(* IEC 61131-3 sources: volt/packages/volt-lsp-iec/test-corpus/lenze-mid/Device/Plc Logic/Application/Library Manager/(unresolved)/cmpopcuastack interfaces, 277 files *)

(* ---- OPCUA_ACTIVATESESSIONREQUEST.dut ---- *)
TYPE OPCUA_ACTIVATESESSIONREQUEST :
STRUCT
	REQUESTHEADER : OpcUa_RequestHeader;
	CLIENTSIGNATURE : OpcUa_SignatureData;
	NOOFCLIENTSOFTWARECERTIFICATES : OpcUa_Int32;
	CLIENTSOFTWARECERTIFICATES : POINTER TO OpcUa_SignedSoftwareCertificate;
	NOOFLOCALEIDS : OpcUa_Int32;
	LOCALEIDS : POINTER TO OpcUa_String;
	USERIDENTITYTOKEN : OpcUa_ExtensionObject;
	USERTOKENSIGNATURE : OpcUa_SignatureData;
END_STRUCT
END_TYPE

(* ---- OPCUA_ACTIVATESESSIONRESPONSE.dut ---- *)
TYPE OPCUA_ACTIVATESESSIONRESPONSE :
STRUCT
	RESPONSEHEADER : OpcUa_ResponseHeader;
	SERVERNONCE : OpcUa_ByteString;
	NOOFRESULTS : OpcUa_Int32;
	RESULTS : POINTER TO OpcUa_StatusCode;
	NOOFDIAGNOSTICINFOS : OpcUa_Int32;
	DIAGNOSTICINFOS : POINTER TO OpcUa_DiagnosticInfo;
END_STRUCT
END_TYPE

(* ---- OPCUA_ADDNODESITEM.dut ---- *)
TYPE OPCUA_ADDNODESITEM :
STRUCT
	PARENTNODEID : OpcUa_ExpandedNodeId;
	REFERENCETYPEID : OpcUa_NodeId;
	REQUESTEDNEWNODEID : OpcUa_ExpandedNodeId;
	BROWSENAME : OpcUa_QualifiedName;
	NODECLASS : OpcUa_NodeClass;
	NODEATTRIBUTES : OpcUa_ExtensionObject;
	TYPEDEFINITION : OpcUa_ExpandedNodeId;
END_STRUCT
END_TYPE

(* ---- OPCUA_ADDNODESREQUEST.dut ---- *)
TYPE OPCUA_ADDNODESREQUEST :
STRUCT
	REQUESTHEADER : OpcUa_RequestHeader;
	NOOFNODESTOADD : OpcUa_Int32;
	NODESTOADD : POINTER TO OpcUa_AddNodesItem;
END_STRUCT
END_TYPE

(* ---- OPCUA_ADDNODESRESPONSE.dut ---- *)
TYPE OPCUA_ADDNODESRESPONSE :
STRUCT
	RESPONSEHEADER : OpcUa_ResponseHeader;
	NOOFRESULTS : OpcUa_Int32;
	RESULTS : POINTER TO OpcUa_AddNodesResult;
	NOOFDIAGNOSTICINFOS : OpcUa_Int32;
	DIAGNOSTICINFOS : POINTER TO OpcUa_DiagnosticInfo;
END_STRUCT
END_TYPE

(* ---- OPCUA_ADDNODESRESULT.dut ---- *)
TYPE OPCUA_ADDNODESRESULT :
STRUCT
	STATUSCODE : OpcUa_StatusCode;
	ADDEDNODEID : OpcUa_NodeId;
END_STRUCT
END_TYPE

(* ---- OPCUA_ADDREFERENCESITEM.dut ---- *)
TYPE OPCUA_ADDREFERENCESITEM :
STRUCT
	SOURCENODEID : OpcUa_NodeId;
	REFERENCETYPEID : OpcUa_NodeId;
	ISFORWARD : OpcUa_Boolean;
	TARGETSERVERURI : OpcUa_String;
	TARGETNODEID : OpcUa_ExpandedNodeId;
	TARGETNODECLASS : OpcUa_NodeClass;
END_STRUCT
END_TYPE

(* ---- OPCUA_ADDREFERENCESREQUEST.dut ---- *)
TYPE OPCUA_ADDREFERENCESREQUEST :
STRUCT
	REQUESTHEADER : OpcUa_RequestHeader;
	NOOFREFERENCESTOADD : OpcUa_Int32;
	REFERENCESTOADD : POINTER TO OpcUa_AddReferencesItem;
END_STRUCT
END_TYPE

(* ---- OPCUA_ADDREFERENCESRESPONSE.dut ---- *)
TYPE OPCUA_ADDREFERENCESRESPONSE :
STRUCT
	RESPONSEHEADER : OpcUa_ResponseHeader;
	NOOFRESULTS : OpcUa_Int32;
	RESULTS : POINTER TO OpcUa_StatusCode;
	NOOFDIAGNOSTICINFOS : OpcUa_Int32;
	DIAGNOSTICINFOS : POINTER TO OpcUa_DiagnosticInfo;
END_STRUCT
END_TYPE

(* ---- OPCUA_AGGREGATECONFIGURATION.dut ---- *)
TYPE OPCUA_AGGREGATECONFIGURATION :
STRUCT
	USESERVERCAPABILITIESDEFAULTS : OpcUa_Boolean;
	TREATUNCERTAINASBAD : OpcUa_Boolean;
	PERCENTDATABAD : OpcUa_Byte;
	PERCENTDATAGOOD : OpcUa_Byte;
	USESLOPEDEXTRAPOLATION : OpcUa_Boolean;
END_STRUCT
END_TYPE

(* ---- OPCUA_AGGREGATEFILTER.dut ---- *)
TYPE OPCUA_AGGREGATEFILTER :
STRUCT
	STARTTIME : OpcUa_DateTime;
	AGGREGATETYPE : OpcUa_NodeId;
	PROCESSINGINTERVAL : OpcUa_Double;
	AGGREGATECONFIGURATION : OpcUa_AggregateConfiguration;
END_STRUCT
END_TYPE

(* ---- OPCUA_AGGREGATEFILTERRESULT.dut ---- *)
TYPE OPCUA_AGGREGATEFILTERRESULT :
STRUCT
	REVISEDSTARTTIME : OpcUa_DateTime;
	REVISEDPROCESSINGINTERVAL : OpcUa_Double;
	REVISEDAGGREGATECONFIGURATION : OpcUa_AggregateConfiguration;
END_STRUCT
END_TYPE

(* ---- OPCUA_ANNOTATION.dut ---- *)
TYPE OPCUA_ANNOTATION :
STRUCT
	MESSAGE : OpcUa_String;
	USERNAME : OpcUa_String;
	ANNOTATIONTIME : OpcUa_DateTime;
END_STRUCT
END_TYPE

(* ---- OPCUA_ANONYMOUSIDENTITYTOKEN.dut ---- *)
TYPE OPCUA_ANONYMOUSIDENTITYTOKEN :
STRUCT
	POLICYID : OpcUa_String;
END_STRUCT
END_TYPE

(* ---- OPCUA_APPLICATIONDESCRIPTION.dut ---- *)
TYPE OPCUA_APPLICATIONDESCRIPTION :
STRUCT
	APPLICATIONURI : OpcUa_String;
	PRODUCTURI : OpcUa_String;
	APPLICATIONNAME : OpcUa_LocalizedText;
	APPLICATIONTYPE : OpcUa_ApplicationType;
	GATEWAYSERVERURI : OpcUa_String;
	DISCOVERYPROFILEURI : OpcUa_String;
	NOOFDISCOVERYURLS : OpcUa_Int32;
	DISCOVERYURLS : POINTER TO OpcUa_String;
END_STRUCT
END_TYPE

(* ---- OPCUA_APPLICATIONTYPE.dut ---- *)
TYPE OPCUA_APPLICATIONTYPE :
(
	OPCUA_APPLICATIONTYPE_SERVER := 0,
	OPCUA_APPLICATIONTYPE_CLIENT := 1,
	OPCUA_APPLICATIONTYPE_CLIENTANDSERVER := 2,
	OPCUA_APPLICATIONTYPE_DISCOVERYSERVER := 3
);
END_TYPE

(* ---- OPCUA_ARGUMENT.dut ---- *)
TYPE OPCUA_ARGUMENT :
STRUCT
	NAME : OpcUa_String;
	DATATYPE : OpcUa_NodeId;
	VALUERANK : OpcUa_Int32;
	NOOFARRAYDIMENSIONS : OpcUa_Int32;
	ARRAYDIMENSIONS : POINTER TO OpcUa_UInt32;
	DESCRIPTION : OpcUa_LocalizedText;
END_STRUCT
END_TYPE

(* ---- OPCUA_ARRAYTYPE.dut ---- *)
TYPE OPCUA_ARRAYTYPE :
(
	OPCUA_VALUERANKS_SCALARORONEDIMENSION := -3,
	OPCUA_VALUERANKS_ANY := -2,
	OPCUA_VALUERANKS_SCALAR := -1,
	OPCUA_VALUERANKS_ONEORMOREDIMENSIONS := 0,
	OPCUA_VALUERANKS_ONEDIMENSION := 1,
	OPCUA_VALUERANKS_TWODIMENSIONS := 2
);
END_TYPE

(* ---- OPCUA_ATTRIBUTEOPERAND.dut ---- *)
TYPE OPCUA_ATTRIBUTEOPERAND :
STRUCT
	NODEID : OpcUa_NodeId;
	ALIAS : OpcUa_String;
	BROWSEPATH : OpcUa_RelativePath;
	ATTRIBUTEID : OpcUa_UInt32;
	INDEXRANGE : OpcUa_String;
END_STRUCT
END_TYPE

(* ---- OPCUA_ATTRIBUTES.dut ---- *)
TYPE OPCUA_ATTRIBUTES :
(
	OPCUA_ATTRIBUTES_NODEID := 1,
	OPCUA_ATTRIBUTES_NODECLASS := 2,
	OPCUA_ATTRIBUTES_BROWSENAME := 3,
	OPCUA_ATTRIBUTES_DISPLAYNAME := 4,
	OPCUA_ATTRIBUTES_DESCRIPTION := 5,
	OPCUA_ATTRIBUTES_WRITEMASK := 6,
	OPCUA_ATTRIBUTES_USERWRITEMASK := 7,
	OPCUA_ATTRIBUTES_ISABSTRACT := 8,
	OPCUA_ATTRIBUTES_SYMMETRIC := 9,
	OPCUA_ATTRIBUTES_INVERSENAME := 10,
	OPCUA_ATTRIBUTES_CONTAINSNOLOOPS := 11,
	OPCUA_ATTRIBUTES_EVENTNOTIFIER := 12,
	OPCUA_ATTRIBUTES_VALUE := 13,
	OPCUA_ATTRIBUTES_DATATYPE := 14,
	OPCUA_ATTRIBUTES_VALUERANK := 15,
	OPCUA_ATTRIBUTES_ARRAYDIMENSIONS := 16,
	OPCUA_ATTRIBUTES_ACCESSLEVEL := 17,
	OPCUA_ATTRIBUTES_USERACCESSLEVEL := 18,
	OPCUA_ATTRIBUTES_MINIMUMSAMPLINGINTERVAL := 19,
	OPCUA_ATTRIBUTES_HISTORIZING := 20,
	OPCUA_ATTRIBUTES_EXECUTABLE := 21,
	OPCUA_ATTRIBUTES_USEREXECUTABLE := 22,
	OPCUA_ATTRIBUTES_DATATYPEDEFINITION := 23,
	OPCUA_ATTRIBUTES_ROLEPERMISSIONS := 24,
	OPCUA_ATTRIBUTES_USERROLEPERMISSIONS := 25,
	OPCUA_ATTRIBUTES_ACCESSRESTRICTIONS := 26,
	OPCUA_ATTRIBUTES_ACCESSLEVELEX := 27
);
END_TYPE

(* ---- OPCUA_AXISINFORMATION.dut ---- *)
TYPE OPCUA_AXISINFORMATION :
STRUCT
	ENGINEERINGUNITS : OpcUa_EUInformation;
	EURANGE : OpcUa_Range;
	TITLE : OpcUa_LocalizedText;
	AXISSCALETYPE : OpcUa_AxisScaleEnumeration;
	NOOFAXISSTEPS : OpcUa_Int32;
	AXISSTEPS : POINTER TO OpcUa_Double;
END_STRUCT
END_TYPE

(* ---- OPCUA_AXISSCALEENUMERATION.dut ---- *)
TYPE OPCUA_AXISSCALEENUMERATION :
(
	OPCUA_AXISSCALEENUMERATION_LINEAR := 0,
	OPCUA_AXISSCALEENUMERATION_LOG := 1,
	OPCUA_AXISSCALEENUMERATION_LN := 2
);
END_TYPE

(* ---- OPCUA_BOOLEAN.dut ---- *)
TYPE OPCUA_BOOLEAN : BOOL;
END_TYPE

(* ---- OPCUA_BROWSEDESCRIPTION.dut ---- *)
TYPE OPCUA_BROWSEDESCRIPTION :
STRUCT
	NODEID : OpcUa_NodeId;
	BROWSEDIRECTION : OpcUa_BrowseDirection;
	REFERENCETYPEID : OpcUa_NodeId;
	INCLUDESUBTYPES : OpcUa_Boolean;
	NODECLASSMASK : OpcUa_UInt32;
	RESULTMASK : OpcUa_UInt32;
END_STRUCT
END_TYPE

(* ---- OPCUA_BROWSEDIRECTION.dut ---- *)
TYPE OPCUA_BROWSEDIRECTION :
(
	OPCUA_BROWSEDIRECTION_FORWARD := 0,
	OPCUA_BROWSEDIRECTION_INVERSE := 1,
	OPCUA_BROWSEDIRECTION_BOTH := 2,
	OPCUA_BROWSEDIRECTION_INVALID := 3
);
END_TYPE

(* ---- OPCUA_BROWSENEXTREQUEST.dut ---- *)
TYPE OPCUA_BROWSENEXTREQUEST :
STRUCT
	REQUESTHEADER : OpcUa_RequestHeader;
	RELEASECONTINUATIONPOINTS : OpcUa_Boolean;
	NOOFCONTINUATIONPOINTS : OpcUa_Int32;
	CONTINUATIONPOINTS : POINTER TO OpcUa_ByteString;
END_STRUCT
END_TYPE

(* ---- OPCUA_BROWSENEXTRESPONSE.dut ---- *)
TYPE OPCUA_BROWSENEXTRESPONSE :
STRUCT
	RESPONSEHEADER : OpcUa_ResponseHeader;
	NOOFRESULTS : OpcUa_Int32;
	RESULTS : POINTER TO OpcUa_BrowseResult;
	NOOFDIAGNOSTICINFOS : OpcUa_Int32;
	DIAGNOSTICINFOS : POINTER TO OpcUa_DiagnosticInfo;
END_STRUCT
END_TYPE

(* ---- OPCUA_BROWSEPATH.dut ---- *)
TYPE OPCUA_BROWSEPATH :
STRUCT
	STARTINGNODE : OpcUa_NodeId;
	RELATIVEPATH : OpcUa_RelativePath;
END_STRUCT
END_TYPE

(* ---- OPCUA_BROWSEPATHRESULT.dut ---- *)
TYPE OPCUA_BROWSEPATHRESULT :
STRUCT
	STATUSCODE : OpcUa_StatusCode;
	NOOFTARGETS : OpcUa_Int32;
	TARGETS : POINTER TO OpcUa_BrowsePathTarget;
END_STRUCT
END_TYPE

(* ---- OPCUA_BROWSEPATHTARGET.dut ---- *)
TYPE OPCUA_BROWSEPATHTARGET :
STRUCT
	TARGETID : OpcUa_ExpandedNodeId;
	REMAININGPATHINDEX : OpcUa_UInt32;
END_STRUCT
END_TYPE

(* ---- OPCUA_BROWSEREQUEST.dut ---- *)
TYPE OPCUA_BROWSEREQUEST :
STRUCT
	REQUESTHEADER : OpcUa_RequestHeader;
	VIEW : OpcUa_ViewDescription;
	REQUESTEDMAXREFERENCESPERNODE : OpcUa_UInt32;
	NOOFNODESTOBROWSE : OpcUa_Int32;
	NODESTOBROWSE : POINTER TO OpcUa_BrowseDescription;
END_STRUCT
END_TYPE

(* ---- OPCUA_BROWSERESPONSE.dut ---- *)
TYPE OPCUA_BROWSERESPONSE :
STRUCT
	RESPONSEHEADER : OpcUa_ResponseHeader;
	NOOFRESULTS : OpcUa_Int32;
	RESULTS : POINTER TO OpcUa_BrowseResult;
	NOOFDIAGNOSTICINFOS : OpcUa_Int32;
	DIAGNOSTICINFOS : POINTER TO OpcUa_DiagnosticInfo;
END_STRUCT
END_TYPE

(* ---- OPCUA_BROWSERESULT.dut ---- *)
TYPE OPCUA_BROWSERESULT :
STRUCT
	STATUSCODE : OpcUa_StatusCode;
	CONTINUATIONPOINT : OpcUa_ByteString;
	NOOFREFERENCES : OpcUa_Int32;
	REFERENCES : POINTER TO OpcUa_ReferenceDescription;
END_STRUCT
END_TYPE

(* ---- OPCUA_BROWSERESULTMASK.dut ---- *)
TYPE OPCUA_BROWSERESULTMASK :
(
	OPCUA_BROWSERESULTMASK_NONE := 0,
	OPCUA_BROWSERESULTMASK_REFERENCETYPEID := 1,
	OPCUA_BROWSERESULTMASK_ISFORWARD := 2,
	OPCUA_BROWSERESULTMASK_NODECLASS := 4,
	OPCUA_BROWSERESULTMASK_BROWSENAME := 8,
	OPCUA_BROWSERESULTMASK_DISPLAYNAME := 16,
	OPCUA_BROWSERESULTMASK_TYPEDEFINITION := 32,
	OPCUA_BROWSERESULTMASK_ALL := 63,
	OPCUA_BROWSERESULTMASK_REFERENCETYPEINFO := 3,
	OPCUA_BROWSERESULTMASK_TARGETINFO := 60
);
END_TYPE

(* ---- OPCUA_BUILDINFO.dut ---- *)
TYPE OPCUA_BUILDINFO :
STRUCT
	PRODUCTURI : OpcUa_String;
	MANUFACTURERNAME : OpcUa_String;
	PRODUCTNAME : OpcUa_String;
	SOFTWAREVERSION : OpcUa_String;
	BUILDNUMBER : OpcUa_String;
	BUILDDATE : OpcUa_DateTime;
END_STRUCT
END_TYPE

(* ---- OPCUA_BUILTINTYPE.dut ---- *)
TYPE OPCUA_BUILTINTYPE :
(
	OPCUATYPE_NULL := 0,
	OPCUATYPE_BOOLEAN := 1,
	OPCUATYPE_SBYTE := 2,
	OPCUATYPE_BYTE := 3,
	OPCUATYPE_INT16 := 4,
	OPCUATYPE_UINT16 := 5,
	OPCUATYPE_INT32 := 6,
	OPCUATYPE_UINT32 := 7,
	OPCUATYPE_INT64 := 8,
	OPCUATYPE_UINT64 := 9,
	OPCUATYPE_FLOAT := 10,
	OPCUATYPE_DOUBLE := 11,
	OPCUATYPE_STRING := 12,
	OPCUATYPE_DATETIME := 13,
	OPCUATYPE_GUID := 14,
	OPCUATYPE_BYTESTRING := 15,
	OPCUATYPE_XMLELEMENT := 16,
	OPCUATYPE_NODEID := 17,
	OPCUATYPE_EXPANDEDNODEID := 18,
	OPCUATYPE_STATUSCODE := 19,
	OPCUATYPE_QUALIFIEDNAME := 20,
	OPCUATYPE_LOCALIZEDTEXT := 21,
	OPCUATYPE_EXTENSIONOBJECT := 22,
	OPCUATYPE_DATAVALUE := 23,
	OPCUATYPE_VARIANT := 24,
	OPCUATYPE_DIAGNOSTICINFO := 25
);
END_TYPE

(* ---- OPCUA_BYTE.dut ---- *)
TYPE OPCUA_BYTE : USINT;
END_TYPE

(* ---- OPCUA_BYTESTRING.dut ---- *)
TYPE OPCUA_BYTESTRING :
STRUCT
	LENGTH : OpcUa_Int32;
	DATA : POINTER TO OpcUa_Byte;
END_STRUCT
END_TYPE

(* ---- OPCUA_CALLMETHODREQUEST.dut ---- *)
TYPE OPCUA_CALLMETHODREQUEST :
STRUCT
	OBJECTID : OpcUa_NodeId;
	METHODID : OpcUa_NodeId;
	NOOFINPUTARGUMENTS : OpcUa_Int32;
	INPUTARGUMENTS : POINTER TO OpcUa_Variant;
END_STRUCT
END_TYPE

(* ---- OPCUA_CALLMETHODRESULT.dut ---- *)
TYPE OPCUA_CALLMETHODRESULT :
STRUCT
	STATUSCODE : OpcUa_StatusCode;
	NOOFINPUTARGUMENTRESULTS : OpcUa_Int32;
	INPUTARGUMENTRESULTS : POINTER TO OpcUa_StatusCode;
	NOOFINPUTARGUMENTDIAGNOSTICINFOS : OpcUa_Int32;
	INPUTARGUMENTDIAGNOSTICINFOS : POINTER TO OpcUa_DiagnosticInfo;
	NOOFOUTPUTARGUMENTS : OpcUa_Int32;
	OUTPUTARGUMENTS : POINTER TO OpcUa_Variant;
END_STRUCT
END_TYPE

(* ---- OPCUA_CALLREQUEST.dut ---- *)
TYPE OPCUA_CALLREQUEST :
STRUCT
	REQUESTHEADER : OpcUa_RequestHeader;
	NOOFMETHODSTOCALL : OpcUa_Int32;
	METHODSTOCALL : POINTER TO OpcUa_CallMethodRequest;
END_STRUCT
END_TYPE

(* ---- OPCUA_CALLRESPONSE.dut ---- *)
TYPE OPCUA_CALLRESPONSE :
STRUCT
	RESPONSEHEADER : OpcUa_ResponseHeader;
	NOOFRESULTS : OpcUa_Int32;
	RESULTS : POINTER TO OpcUa_CallMethodResult;
	NOOFDIAGNOSTICINFOS : OpcUa_Int32;
	DIAGNOSTICINFOS : POINTER TO OpcUa_DiagnosticInfo;
END_STRUCT
END_TYPE

(* ---- OPCUA_CANCELREQUEST.dut ---- *)
TYPE OPCUA_CANCELREQUEST :
STRUCT
	REQUESTHEADER : OpcUa_RequestHeader;
	REQUESTHANDLE : OpcUa_UInt32;
END_STRUCT
END_TYPE

(* ---- OPCUA_CANCELRESPONSE.dut ---- *)
TYPE OPCUA_CANCELRESPONSE :
STRUCT
	RESPONSEHEADER : OpcUa_ResponseHeader;
	CANCELCOUNT : OpcUa_UInt32;
END_STRUCT
END_TYPE

(* ---- OPCUA_CHANNELSECURITYTOKEN.dut ---- *)
TYPE OPCUA_CHANNELSECURITYTOKEN :
STRUCT
	CHANNELID : OpcUa_UInt32;
	TOKENID : OpcUa_UInt32;
	CREATEDAT : OpcUa_DateTime;
	REVISEDLIFETIME : OpcUa_UInt32;
END_STRUCT
END_TYPE

(* ---- OPCUA_CHARA.dut ---- *)
TYPE OPCUA_CHARA : BYTE;
END_TYPE

(* ---- OPCUA_CLOSESECURECHANNELREQUEST.dut ---- *)
TYPE OPCUA_CLOSESECURECHANNELREQUEST :
STRUCT
	REQUESTHEADER : OpcUa_RequestHeader;
END_STRUCT
END_TYPE

(* ---- OPCUA_CLOSESECURECHANNELRESPONSE.dut ---- *)
TYPE OPCUA_CLOSESECURECHANNELRESPONSE :
STRUCT
	RESPONSEHEADER : OpcUa_ResponseHeader;
END_STRUCT
END_TYPE

(* ---- OPCUA_CLOSESESSIONREQUEST.dut ---- *)
TYPE OPCUA_CLOSESESSIONREQUEST :
STRUCT
	REQUESTHEADER : OpcUa_RequestHeader;
	DELETESUBSCRIPTIONS : OpcUa_Boolean;
END_STRUCT
END_TYPE

(* ---- OPCUA_CLOSESESSIONRESPONSE.dut ---- *)
TYPE OPCUA_CLOSESESSIONRESPONSE :
STRUCT
	RESPONSEHEADER : OpcUa_ResponseHeader;
END_STRUCT
END_TYPE

(* ---- OPCUA_COMPLEXNUMBERTYPE.dut ---- *)
TYPE OPCUA_COMPLEXNUMBERTYPE :
STRUCT
	REAL_CDS : OpcUa_Float;
	IMAGINARY : OpcUa_Float;
END_STRUCT
END_TYPE

(* ---- OPCUA_CONTENTFILTER.dut ---- *)
TYPE OPCUA_CONTENTFILTER :
STRUCT
	NOOFELEMENTS : OpcUa_Int32;
	ELEMENTS : POINTER TO OpcUa_ContentFilterElement;
END_STRUCT
END_TYPE

(* ---- OPCUA_CONTENTFILTERELEMENT.dut ---- *)
TYPE OPCUA_CONTENTFILTERELEMENT :
STRUCT
	FILTEROPERATOR : OpcUa_FilterOperator;
	NOOFFILTEROPERANDS : OpcUa_Int32;
	FILTEROPERANDS : POINTER TO OpcUa_ExtensionObject;
END_STRUCT
END_TYPE

(* ---- OPCUA_CONTENTFILTERELEMENTRESULT.dut ---- *)
TYPE OPCUA_CONTENTFILTERELEMENTRESULT :
STRUCT
	STATUSCODE : OpcUa_StatusCode;
	NOOFOPERANDSTATUSCODES : OpcUa_Int32;
	OPERANDSTATUSCODES : POINTER TO OpcUa_StatusCode;
	NOOFOPERANDDIAGNOSTICINFOS : OpcUa_Int32;
	OPERANDDIAGNOSTICINFOS : POINTER TO OpcUa_DiagnosticInfo;
END_STRUCT
END_TYPE

(* ---- OPCUA_CONTENTFILTERRESULT.dut ---- *)
TYPE OPCUA_CONTENTFILTERRESULT :
STRUCT
	NOOFELEMENTRESULTS : OpcUa_Int32;
	ELEMENTRESULTS : POINTER TO OpcUa_ContentFilterElementResult;
	NOOFELEMENTDIAGNOSTICINFOS : OpcUa_Int32;
	ELEMENTDIAGNOSTICINFOS : POINTER TO OpcUa_DiagnosticInfo;
END_STRUCT
END_TYPE

(* ---- OPCUA_CREATEMONITOREDITEMSREQUEST.dut ---- *)
TYPE OPCUA_CREATEMONITOREDITEMSREQUEST :
STRUCT
	REQUESTHEADER : OpcUa_RequestHeader;
	SUBSCRIPTIONID : OpcUa_UInt32;
	TIMESTAMPSTORETURN : OpcUa_TimestampsToReturn;
	NOOFITEMSTOCREATE : OpcUa_Int32;
	ITEMSTOCREATE : POINTER TO OpcUa_MonitoredItemCreateRequest;
END_STRUCT
END_TYPE

(* ---- OPCUA_CREATEMONITOREDITEMSRESPONSE.dut ---- *)
TYPE OPCUA_CREATEMONITOREDITEMSRESPONSE :
STRUCT
	RESPONSEHEADER : OpcUa_ResponseHeader;
	NOOFRESULTS : OpcUa_Int32;
	RESULTS : POINTER TO OpcUa_MonitoredItemCreateResult;
	NOOFDIAGNOSTICINFOS : OpcUa_Int32;
	DIAGNOSTICINFOS : POINTER TO OpcUa_DiagnosticInfo;
END_STRUCT
END_TYPE

(* ---- OPCUA_CREATESESSIONREQUEST.dut ---- *)
TYPE OPCUA_CREATESESSIONREQUEST :
STRUCT
	REQUESTHEADER : OpcUa_RequestHeader;
	CLIENTDESCRIPTION : OpcUa_ApplicationDescription;
	SERVERURI : OpcUa_String;
	ENDPOINTURL : OpcUa_String;
	SESSIONNAME : OpcUa_String;
	CLIENTNONCE : OpcUa_ByteString;
	CLIENTCERTIFICATE : OpcUa_ByteString;
	REQUESTEDSESSIONTIMEOUT : OpcUa_Double;
	MAXRESPONSEMESSAGESIZE : OpcUa_UInt32;
END_STRUCT
END_TYPE

(* ---- OPCUA_CREATESESSIONRESPONSE.dut ---- *)
TYPE OPCUA_CREATESESSIONRESPONSE :
STRUCT
	RESPONSEHEADER : OpcUa_ResponseHeader;
	SESSIONID : OpcUa_NodeId;
	AUTHENTICATIONTOKEN : OpcUa_NodeId;
	REVISEDSESSIONTIMEOUT : OpcUa_Double;
	SERVERNONCE : OpcUa_ByteString;
	SERVERCERTIFICATE : OpcUa_ByteString;
	NOOFSERVERENDPOINTS : OpcUa_Int32;
	SERVERENDPOINTS : POINTER TO OpcUa_EndpointDescription;
	NOOFSERVERSOFTWARECERTIFICATES : OpcUa_Int32;
	SERVERSOFTWARECERTIFICATES : POINTER TO OpcUa_SignedSoftwareCertificate;
	SERVERSIGNATURE : OpcUa_SignatureData;
	MAXREQUESTMESSAGESIZE : OpcUa_UInt32;
END_STRUCT
END_TYPE

(* ---- OPCUA_CREATESUBSCRIPTIONREQUEST.dut ---- *)
TYPE OPCUA_CREATESUBSCRIPTIONREQUEST :
STRUCT
	REQUESTHEADER : OpcUa_RequestHeader;
	REQUESTEDPUBLISHINGINTERVAL : OpcUa_Double;
	REQUESTEDLIFETIMECOUNT : OpcUa_UInt32;
	REQUESTEDMAXKEEPALIVECOUNT : OpcUa_UInt32;
	MAXNOTIFICATIONSPERPUBLISH : OpcUa_UInt32;
	PUBLISHINGENABLED : OpcUa_Boolean;
	PRIORITY : OpcUa_Byte;
END_STRUCT
END_TYPE

(* ---- OPCUA_CREATESUBSCRIPTIONRESPONSE.dut ---- *)
TYPE OPCUA_CREATESUBSCRIPTIONRESPONSE :
STRUCT
	RESPONSEHEADER : OpcUa_ResponseHeader;
	SUBSCRIPTIONID : OpcUa_UInt32;
	REVISEDPUBLISHINGINTERVAL : OpcUa_Double;
	REVISEDLIFETIMECOUNT : OpcUa_UInt32;
	REVISEDMAXKEEPALIVECOUNT : OpcUa_UInt32;
END_STRUCT
END_TYPE

(* ---- OPCUA_CRYPTOPROVIDER.dut ---- *)
TYPE OPCUA_CRYPTOPROVIDER :
STRUCT
END_STRUCT
END_TYPE

(* ---- OPCUA_CRYPTOPROVIDER_CONFIG.dut ---- *)
TYPE OPCUA_CRYPTOPROVIDER_CONFIG :
STRUCT
	NAME : POINTER TO STRING;
	NONCESIZE : OpcUa_UInt32;
	SYMMETRICSIGNATUREKEYSIZE : OpcUa_UInt32;
	SYMMETRICSIGNATURESIZE : OpcUa_UInt32;
	SYMMETRICENCRYPTIONKEYSIZE : OpcUa_UInt32;
	SYMMETRICENCRYPTIONBLOCKSIZE : OpcUa_UInt32;
	SYMMETRICENCRYPTIONIVSIZE : OpcUa_UInt32;
	ASYMMETRICENCRYPTIONOVERHEAD : OpcUa_UInt32;
	MAXIMUMASYMMETRICKEYLENGTH : OpcUa_UInt32;
	MINIMUMASYMMETRICKEYLENGTH : OpcUa_UInt32;
	ASYMMETRICSIGNATUREURI : POINTER TO STRING;
	ASYMMETRICENCRYPTIONURI : POINTER TO STRING;
	SYMMETRICSIGNATUREURI : POINTER TO STRING;
	SYMMETRICENCRYPTIONURI : POINTER TO STRING;
END_STRUCT
END_TYPE

(* ---- OPCUA_DATACHANGEFILTER.dut ---- *)
TYPE OPCUA_DATACHANGEFILTER :
STRUCT
	TRIGGER : OpcUa_DataChangeTrigger;
	DEADBANDTYPE : OpcUa_UInt32;
	DEADBANDVALUE : OpcUa_Double;
END_STRUCT
END_TYPE

(* ---- OPCUA_DATACHANGENOTIFICATION.dut ---- *)
TYPE OPCUA_DATACHANGENOTIFICATION :
STRUCT
	NOOFMONITOREDITEMS : OpcUa_Int32;
	MONITOREDITEMS : POINTER TO OpcUa_MonitoredItemNotification;
	NOOFDIAGNOSTICINFOS : OpcUa_Int32;
	DIAGNOSTICINFOS : POINTER TO OpcUa_DiagnosticInfo;
END_STRUCT
END_TYPE

(* ---- OPCUA_DATACHANGETRIGGER.dut ---- *)
TYPE OPCUA_DATACHANGETRIGGER :
(
	OPCUA_DATACHANGETRIGGER_STATUS := 0,
	OPCUA_DATACHANGETRIGGER_STATUSVALUE := 1,
	OPCUA_DATACHANGETRIGGER_STATUSVALUETIMESTAMP := 2
);
END_TYPE

(* ---- OPCUA_DATATYPEATTRIBUTES.dut ---- *)
TYPE OPCUA_DATATYPEATTRIBUTES :
STRUCT
	SPECIFIEDATTRIBUTES : OpcUa_UInt32;
	DISPLAYNAME : OpcUa_LocalizedText;
	DESCRIPTION : OpcUa_LocalizedText;
	WRITEMASK : OpcUa_UInt32;
	USERWRITEMASK : OpcUa_UInt32;
	ISABSTRACT : OpcUa_Boolean;
END_STRUCT
END_TYPE

(* ---- OPCUA_DATAVALUE.dut ---- *)
TYPE OPCUA_DATAVALUE :
STRUCT
	VALUE : OpcUa_Variant;
	STATUSCODE : OpcUa_StatusCode;
	SOURCETIMESTAMP : OpcUa_DateTime;
	SERVERTIMESTAMP : OpcUa_DateTime;
	SOURCEPICOSECONDS : OpcUa_UInt16;
	SERVERPICOSECONDS : OpcUa_UInt16;
END_STRUCT
END_TYPE

(* ---- OPCUA_DATETIME.dut ---- *)
TYPE OPCUA_DATETIME : LINT;
END_TYPE

(* ---- OPCUA_DECODER.dut ---- *)
TYPE OPCUA_DECODER :
STRUCT
END_STRUCT
END_TYPE

(* ---- OPCUA_DELETEATTIMEDETAILS.dut ---- *)
TYPE OPCUA_DELETEATTIMEDETAILS :
STRUCT
	NODEID : OpcUa_NodeId;
	NOOFREQTIMES : OpcUa_Int32;
	REQTIMES : POINTER TO OpcUa_DateTime;
END_STRUCT
END_TYPE

(* ---- OPCUA_DELETEEVENTDETAILS.dut ---- *)
TYPE OPCUA_DELETEEVENTDETAILS :
STRUCT
	NODEID : OpcUa_NodeId;
	NOOFEVENTIDS : OpcUa_Int32;
	EVENTIDS : POINTER TO OpcUa_ByteString;
END_STRUCT
END_TYPE

(* ---- OPCUA_DELETEMONITOREDITEMSREQUEST.dut ---- *)
TYPE OPCUA_DELETEMONITOREDITEMSREQUEST :
STRUCT
	REQUESTHEADER : OpcUa_RequestHeader;
	SUBSCRIPTIONID : OpcUa_UInt32;
	NOOFMONITOREDITEMIDS : OpcUa_Int32;
	MONITOREDITEMIDS : POINTER TO OpcUa_UInt32;
END_STRUCT
END_TYPE

(* ---- OPCUA_DELETEMONITOREDITEMSRESPONSE.dut ---- *)
TYPE OPCUA_DELETEMONITOREDITEMSRESPONSE :
STRUCT
	RESPONSEHEADER : OpcUa_ResponseHeader;
	NOOFRESULTS : OpcUa_Int32;
	RESULTS : POINTER TO OpcUa_StatusCode;
	NOOFDIAGNOSTICINFOS : OpcUa_Int32;
	DIAGNOSTICINFOS : POINTER TO OpcUa_DiagnosticInfo;
END_STRUCT
END_TYPE

(* ---- OPCUA_DELETENODESITEM.dut ---- *)
TYPE OPCUA_DELETENODESITEM :
STRUCT
	NODEID : OpcUa_NodeId;
	DELETETARGETREFERENCES : OpcUa_Boolean;
END_STRUCT
END_TYPE

(* ---- OPCUA_DELETENODESREQUEST.dut ---- *)
TYPE OPCUA_DELETENODESREQUEST :
STRUCT
	REQUESTHEADER : OpcUa_RequestHeader;
	NOOFNODESTODELETE : OpcUa_Int32;
	NODESTODELETE : POINTER TO OpcUa_DeleteNodesItem;
END_STRUCT
END_TYPE

(* ---- OPCUA_DELETENODESRESPONSE.dut ---- *)
TYPE OPCUA_DELETENODESRESPONSE :
STRUCT
	RESPONSEHEADER : OpcUa_ResponseHeader;
	NOOFRESULTS : OpcUa_Int32;
	RESULTS : POINTER TO OpcUa_StatusCode;
	NOOFDIAGNOSTICINFOS : OpcUa_Int32;
	DIAGNOSTICINFOS : POINTER TO OpcUa_DiagnosticInfo;
END_STRUCT
END_TYPE

(* ---- OPCUA_DELETERAWMODIFIEDDETAILS.dut ---- *)
TYPE OPCUA_DELETERAWMODIFIEDDETAILS :
STRUCT
	NODEID : OpcUa_NodeId;
	ISDELETEMODIFIED : OpcUa_Boolean;
	STARTTIME : OpcUa_DateTime;
	ENDTIME : OpcUa_DateTime;
END_STRUCT
END_TYPE

(* ---- OPCUA_DELETEREFERENCESITEM.dut ---- *)
TYPE OPCUA_DELETEREFERENCESITEM :
STRUCT
	SOURCENODEID : OpcUa_NodeId;
	REFERENCETYPEID : OpcUa_NodeId;
	ISFORWARD : OpcUa_Boolean;
	TARGETNODEID : OpcUa_ExpandedNodeId;
	DELETEBIDIRECTIONAL : OpcUa_Boolean;
END_STRUCT
END_TYPE

(* ---- OPCUA_DELETEREFERENCESREQUEST.dut ---- *)
TYPE OPCUA_DELETEREFERENCESREQUEST :
STRUCT
	REQUESTHEADER : OpcUa_RequestHeader;
	NOOFREFERENCESTODELETE : OpcUa_Int32;
	REFERENCESTODELETE : POINTER TO OpcUa_DeleteReferencesItem;
END_STRUCT
END_TYPE

(* ---- OPCUA_DELETEREFERENCESRESPONSE.dut ---- *)
TYPE OPCUA_DELETEREFERENCESRESPONSE :
STRUCT
	RESPONSEHEADER : OpcUa_ResponseHeader;
	NOOFRESULTS : OpcUa_Int32;
	RESULTS : POINTER TO OpcUa_StatusCode;
	NOOFDIAGNOSTICINFOS : OpcUa_Int32;
	DIAGNOSTICINFOS : POINTER TO OpcUa_DiagnosticInfo;
END_STRUCT
END_TYPE

(* ---- OPCUA_DELETESUBSCRIPTIONSREQUEST.dut ---- *)
TYPE OPCUA_DELETESUBSCRIPTIONSREQUEST :
STRUCT
	REQUESTHEADER : OpcUa_RequestHeader;
	NOOFSUBSCRIPTIONIDS : OpcUa_Int32;
	SUBSCRIPTIONIDS : POINTER TO OpcUa_UInt32;
END_STRUCT
END_TYPE

(* ---- OPCUA_DELETESUBSCRIPTIONSRESPONSE.dut ---- *)
TYPE OPCUA_DELETESUBSCRIPTIONSRESPONSE :
STRUCT
	RESPONSEHEADER : OpcUa_ResponseHeader;
	NOOFRESULTS : OpcUa_Int32;
	RESULTS : POINTER TO OpcUa_StatusCode;
	NOOFDIAGNOSTICINFOS : OpcUa_Int32;
	DIAGNOSTICINFOS : POINTER TO OpcUa_DiagnosticInfo;
END_STRUCT
END_TYPE

(* ---- OPCUA_DIAGNOSTICINFO.dut ---- *)
TYPE OPCUA_DIAGNOSTICINFO :
STRUCT
	SYMBOLICID : OpcUa_Int32;
	NAMESPACEURI : OpcUa_Int32;
	LOCALE : OpcUa_Int32;
	LOCALIZEDTEXT : OpcUa_Int32;
	ADDITIONALINFO : OpcUa_String;
	INNERSTATUSCODE : OpcUa_StatusCode;
	INNERDIAGNOSTICINFO : POINTER TO OpcUa_DiagnosticInfo;
END_STRUCT
END_TYPE

(* ---- OPCUA_DOUBLE.dut ---- *)
TYPE OPCUA_DOUBLE : LREAL;
END_TYPE

(* ---- OPCUA_DOUBLECOMPLEXNUMBERTYPE.dut ---- *)
TYPE OPCUA_DOUBLECOMPLEXNUMBERTYPE :
STRUCT
	REAL_CDS : OpcUa_Double;
	IMAGINARY : OpcUa_Double;
END_STRUCT
END_TYPE

(* ---- OPCUA_ELEMENTOPERAND.dut ---- *)
TYPE OPCUA_ELEMENTOPERAND :
STRUCT
	INDEX : OpcUa_UInt32;
END_STRUCT
END_TYPE

(* ---- OPCUA_ENCODEABLEOBJECTBODY.dut ---- *)
TYPE OPCUA_ENCODEABLEOBJECTBODY :
STRUCT
	OBJECT : POINTER TO BYTE;
	TYPE_CDS : POINTER TO OpcUa_EncodeableType;
END_STRUCT
END_TYPE

(* ---- OPCUA_ENCODEABLETYPE.dut ---- *)
TYPE OPCUA_ENCODEABLETYPE :
STRUCT
END_STRUCT
END_TYPE

(* ---- OPCUA_ENCODER.dut ---- *)
TYPE OPCUA_ENCODER :
STRUCT
END_STRUCT
END_TYPE

(* ---- OPCUA_ENDPOINTCONFIGURATION.dut ---- *)
TYPE OPCUA_ENDPOINTCONFIGURATION :
STRUCT
	OPERATIONTIMEOUT : OpcUa_Int32;
	USEBINARYENCODING : OpcUa_Boolean;
	MAXSTRINGLENGTH : OpcUa_Int32;
	MAXBYTESTRINGLENGTH : OpcUa_Int32;
	MAXARRAYLENGTH : OpcUa_Int32;
	MAXMESSAGESIZE : OpcUa_Int32;
	MAXBUFFERSIZE : OpcUa_Int32;
	CHANNELLIFETIME : OpcUa_Int32;
	SECURITYTOKENLIFETIME : OpcUa_Int32;
END_STRUCT
END_TYPE

(* ---- OPCUA_ENDPOINTDESCRIPTION.dut ---- *)
TYPE OPCUA_ENDPOINTDESCRIPTION :
STRUCT
	ENDPOINTURL : OpcUa_String;
	SERVER : OpcUa_ApplicationDescription;
	SERVERCERTIFICATE : OpcUa_ByteString;
	SECURITYMODE : OpcUa_MessageSecurityMode;
	SECURITYPOLICYURI : OpcUa_String;
	NOOFUSERIDENTITYTOKENS : OpcUa_Int32;
	USERIDENTITYTOKENS : POINTER TO OpcUa_UserTokenPolicy;
	TRANSPORTPROFILEURI : OpcUa_String;
	SECURITYLEVEL : OpcUa_Byte;
END_STRUCT
END_TYPE

(* ---- OPCUA_ENDPOINTURLLISTDATATYPE.dut ---- *)
TYPE OPCUA_ENDPOINTURLLISTDATATYPE :
STRUCT
	NOOFENDPOINTURLLIST : OpcUa_Int32;
	ENDPOINTURLLIST : POINTER TO OpcUa_String;
END_STRUCT
END_TYPE

(* ---- OPCUA_ENUMDEFINITION.dut ---- *)
TYPE OPCUA_ENUMDEFINITION :
STRUCT
	NOOFFIELDS : OpcUa_Int32;
	FIELDS : POINTER TO OpcUa_EnumField;
END_STRUCT
END_TYPE

(* ---- OPCUA_ENUMFIELD.dut ---- *)
TYPE OPCUA_ENUMFIELD :
STRUCT
	VALUE : OpcUa_Int64;
	DISPLAYNAME : OpcUa_LocalizedText;
	DESCRIPTION : OpcUa_LocalizedText;
	NAME : OpcUa_String;
END_STRUCT
END_TYPE

(* ---- OPCUA_ENUMVALUETYPE.dut ---- *)
TYPE OPCUA_ENUMVALUETYPE :
STRUCT
	VALUE : OpcUa_Int64;
	DISPLAYNAME : OpcUa_LocalizedText;
	DESCRIPTION : OpcUa_LocalizedText;
END_STRUCT
END_TYPE

(* ---- OPCUA_EUINFORMATION.dut ---- *)
TYPE OPCUA_EUINFORMATION :
STRUCT
	NAMESPACEURI : OpcUa_String;
	UNITID : OpcUa_Int32;
	DISPLAYNAME : OpcUa_LocalizedText;
	DESCRIPTION : OpcUa_LocalizedText;
END_STRUCT
END_TYPE

(* ---- OPCUA_EVENTFIELDLIST.dut ---- *)
TYPE OPCUA_EVENTFIELDLIST :
STRUCT
	CLIENTHANDLE : OpcUa_UInt32;
	NOOFEVENTFIELDS : OpcUa_Int32;
	EVENTFIELDS : POINTER TO OpcUa_Variant;
END_STRUCT
END_TYPE

(* ---- OPCUA_EVENTFILTER.dut ---- *)
TYPE OPCUA_EVENTFILTER :
STRUCT
	NOOFSELECTCLAUSES : OpcUa_Int32;
	SELECTCLAUSES : POINTER TO OpcUa_SimpleAttributeOperand;
	WHERECLAUSE : OpcUa_ContentFilter;
END_STRUCT
END_TYPE

(* ---- OPCUA_EVENTFILTERRESULT.dut ---- *)
TYPE OPCUA_EVENTFILTERRESULT :
STRUCT
	NOOFSELECTCLAUSERESULTS : OpcUa_Int32;
	SELECTCLAUSERESULTS : POINTER TO OpcUa_StatusCode;
	NOOFSELECTCLAUSEDIAGNOSTICINFOS : OpcUa_Int32;
	SELECTCLAUSEDIAGNOSTICINFOS : POINTER TO OpcUa_DiagnosticInfo;
	WHERECLAUSERESULT : OpcUa_ContentFilterResult;
END_STRUCT
END_TYPE

(* ---- OPCUA_EVENTNOTIFICATIONLIST.dut ---- *)
TYPE OPCUA_EVENTNOTIFICATIONLIST :
STRUCT
	NOOFEVENTS : OpcUa_Int32;
	EVENTS : POINTER TO OpcUa_EventFieldList;
END_STRUCT
END_TYPE

(* ---- OPCUA_EXPANDEDNODEID.dut ---- *)
TYPE OPCUA_EXPANDEDNODEID :
STRUCT
	NODEID : OpcUa_NodeId;
	NAMESPACEURI : OpcUa_String;
	SERVERINDEX : OpcUa_UInt32;
END_STRUCT
END_TYPE

(* ---- OPCUA_EXTENSIONOBJECT.dut ---- *)
TYPE OPCUA_EXTENSIONOBJECT :
STRUCT
	TYPEID : OpcUa_ExpandedNodeId;
	ENCODING : OpcUa_ExtensionObjectEncoding;
	BODY : OpcUa_ExtensionObject_Body;
	BODYSIZE : OpcUa_Int32;
END_STRUCT
END_TYPE

(* ---- OPCUA_EXTENSIONOBJECT_BODY.dut ---- *)
TYPE OPCUA_EXTENSIONOBJECT_BODY :
UNION
	BINARY : OpcUa_ByteString;
	XML : OpcUa_ByteString;
	ENCODEABLEOBJECT : OpcUa_EncodeableObjectBody;
END_UNION
END_TYPE

(* ---- OPCUA_EXTENSIONOBJECTENCODING.dut ---- *)
TYPE OPCUA_EXTENSIONOBJECTENCODING :
(
	OPCUA_EXTENSIONOBJECTENCODING_NONE := 0,
	OPCUA_EXTENSIONOBJECTENCODING_BINARY := 1,
	OPCUA_EXTENSIONOBJECTENCODING_XML := 2,
	OPCUA_EXTENSIONOBJECTENCODING_ENCODEABLEOBJECT := 3
);
END_TYPE

(* ---- OPCUA_FILTEROPERATOR.dut ---- *)
TYPE OPCUA_FILTEROPERATOR :
(
	OPCUA_FILTEROPERATOR_EQUALS := 0,
	OPCUA_FILTEROPERATOR_ISNULL := 1,
	OPCUA_FILTEROPERATOR_GREATERTHAN := 2,
	OPCUA_FILTEROPERATOR_LESSTHAN := 3,
	OPCUA_FILTEROPERATOR_GREATERTHANOREQUAL := 4,
	OPCUA_FILTEROPERATOR_LESSTHANOREQUAL := 5,
	OPCUA_FILTEROPERATOR_LIKE := 6,
	OPCUA_FILTEROPERATOR_NOT := 7,
	OPCUA_FILTEROPERATOR_BETWEEN := 8,
	OPCUA_FILTEROPERATOR_INLIST := 9,
	OPCUA_FILTEROPERATOR_AND := 10,
	OPCUA_FILTEROPERATOR_OR := 11,
	OPCUA_FILTEROPERATOR_CAST := 12,
	OPCUA_FILTEROPERATOR_INVIEW := 13,
	OPCUA_FILTEROPERATOR_OFTYPE := 14,
	OPCUA_FILTEROPERATOR_RELATEDTO := 15,
	OPCUA_FILTEROPERATOR_BITWISEAND := 16,
	OPCUA_FILTEROPERATOR_BITWISEOR := 17
);
END_TYPE

(* ---- OPCUA_FINDSERVERSONNETWORKREQUEST.dut ---- *)
TYPE OPCUA_FINDSERVERSONNETWORKREQUEST :
STRUCT
	REQUESTHEADER : OpcUa_RequestHeader;
	STARTINGRECORDID : OpcUa_UInt32;
	MAXRECORDSTORETURN : OpcUa_UInt32;
	NOOFSERVERCAPABILITYFILTER : OpcUa_Int32;
	SERVERCAPABILITYFILTER : POINTER TO OpcUa_String;
END_STRUCT
END_TYPE

(* ---- OPCUA_FINDSERVERSONNETWORKRESPONSE.dut ---- *)
TYPE OPCUA_FINDSERVERSONNETWORKRESPONSE :
STRUCT
	RESPONSEHEADER : OpcUa_ResponseHeader;
	LASTCOUNTERRESETTIME : OpcUa_DateTime;
	NOOFSERVERS : OpcUa_Int32;
	SERVERS : POINTER TO OpcUa_ServerOnNetwork;
END_STRUCT
END_TYPE

(* ---- OPCUA_FINDSERVERSREQUEST.dut ---- *)
TYPE OPCUA_FINDSERVERSREQUEST :
STRUCT
	REQUESTHEADER : OpcUa_RequestHeader;
	ENDPOINTURL : OpcUa_String;
	NOOFLOCALEIDS : OpcUa_Int32;
	LOCALEIDS : POINTER TO OpcUa_String;
	NOOFSERVERURIS : OpcUa_Int32;
	SERVERURIS : POINTER TO OpcUa_String;
END_STRUCT
END_TYPE

(* ---- OPCUA_FINDSERVERSRESPONSE.dut ---- *)
TYPE OPCUA_FINDSERVERSRESPONSE :
STRUCT
	RESPONSEHEADER : OpcUa_ResponseHeader;
	NOOFSERVERS : OpcUa_Int32;
	SERVERS : POINTER TO OpcUa_ApplicationDescription;
END_STRUCT
END_TYPE

(* ---- OPCUA_FLOAT.dut ---- *)
TYPE OPCUA_FLOAT : REAL;
END_TYPE

(* ---- OPCUA_GENERICATTRIBUTES.dut ---- *)
TYPE OPCUA_GENERICATTRIBUTES :
STRUCT
	SPECIFIEDATTRIBUTES : OpcUa_UInt32;
	DISPLAYNAME : OpcUa_LocalizedText;
	DESCRIPTION : OpcUa_LocalizedText;
	WRITEMASK : OpcUa_UInt32;
	USERWRITEMASK : OpcUa_UInt32;
	NOOFATTRIBUTEVALUES : OpcUa_Int32;
	ATTRIBUTEVALUES : POINTER TO OpcUa_GenericAttributeValue;
END_STRUCT
END_TYPE

(* ---- OPCUA_GENERICATTRIBUTEVALUE.dut ---- *)
TYPE OPCUA_GENERICATTRIBUTEVALUE :
STRUCT
	ATTRIBUTEID : OpcUa_UInt32;
	VALUE : OpcUa_Variant;
END_STRUCT
END_TYPE

(* ---- OPCUA_GETENDPOINTSREQUEST.dut ---- *)
TYPE OPCUA_GETENDPOINTSREQUEST :
STRUCT
	REQUESTHEADER : OpcUa_RequestHeader;
	ENDPOINTURL : OpcUa_String;
	NOOFLOCALEIDS : OpcUa_Int32;
	LOCALEIDS : POINTER TO OpcUa_String;
	NOOFPROFILEURIS : OpcUa_Int32;
	PROFILEURIS : POINTER TO OpcUa_String;
END_STRUCT
END_TYPE

(* ---- OPCUA_GETENDPOINTSRESPONSE.dut ---- *)
TYPE OPCUA_GETENDPOINTSRESPONSE :
STRUCT
	RESPONSEHEADER : OpcUa_ResponseHeader;
	NOOFENDPOINTS : OpcUa_Int32;
	ENDPOINTS : POINTER TO OpcUa_EndpointDescription;
END_STRUCT
END_TYPE

(* ---- OPCUA_GUID.dut ---- *)
TYPE OPCUA_GUID :
STRUCT
	DATA1 : OpcUa_UInt32;
	DATA2 : OpcUa_UInt16;
	DATA3 : OpcUa_UInt16;
	DATA4 : ARRAY [0..7] OF OpcUa_Byte;
END_STRUCT
END_TYPE

(* ---- OPCUA_HANDLE.dut ---- *)
TYPE OPCUA_HANDLE : POINTER TO BYTE;
END_TYPE

(* ---- OPCUA_HISTORYDATA.dut ---- *)
TYPE OPCUA_HISTORYDATA :
STRUCT
	NOOFDATAVALUES : OpcUa_Int32;
	DATAVALUES : POINTER TO OpcUa_DataValue;
END_STRUCT
END_TYPE

(* ---- OPCUA_HISTORYEVENT.dut ---- *)
TYPE OPCUA_HISTORYEVENT :
STRUCT
	NOOFEVENTS : OpcUa_Int32;
	EVENTS : POINTER TO OpcUa_HistoryEventFieldList;
END_STRUCT
END_TYPE

(* ---- OPCUA_HISTORYEVENTFIELDLIST.dut ---- *)
TYPE OPCUA_HISTORYEVENTFIELDLIST :
STRUCT
	NOOFEVENTFIELDS : OpcUa_Int32;
	EVENTFIELDS : POINTER TO OpcUa_Variant;
END_STRUCT
END_TYPE

(* ---- OPCUA_HISTORYMODIFIEDDATA.dut ---- *)
TYPE OPCUA_HISTORYMODIFIEDDATA :
STRUCT
	NOOFDATAVALUES : OpcUa_Int32;
	DATAVALUES : POINTER TO OpcUa_DataValue;
	NOOFMODIFICATIONINFOS : OpcUa_Int32;
	MODIFICATIONINFOS : POINTER TO OpcUa_ModificationInfo;
END_STRUCT
END_TYPE

(* ---- OPCUA_HISTORYREADREQUEST.dut ---- *)
TYPE OPCUA_HISTORYREADREQUEST :
STRUCT
	REQUESTHEADER : OpcUa_RequestHeader;
	HISTORYREADDETAILS : OpcUa_ExtensionObject;
	TIMESTAMPSTORETURN : OpcUa_TimestampsToReturn;
	RELEASECONTINUATIONPOINTS : OpcUa_Boolean;
	NOOFNODESTOREAD : OpcUa_Int32;
	NODESTOREAD : POINTER TO OpcUa_HistoryReadValueId;
END_STRUCT
END_TYPE

(* ---- OPCUA_HISTORYREADRESPONSE.dut ---- *)
TYPE OPCUA_HISTORYREADRESPONSE :
STRUCT
	RESPONSEHEADER : OpcUa_ResponseHeader;
	NOOFRESULTS : OpcUa_Int32;
	RESULTS : POINTER TO OpcUa_HistoryReadResult;
	NOOFDIAGNOSTICINFOS : OpcUa_Int32;
	DIAGNOSTICINFOS : POINTER TO OpcUa_DiagnosticInfo;
END_STRUCT
END_TYPE

(* ---- OPCUA_HISTORYREADRESULT.dut ---- *)
TYPE OPCUA_HISTORYREADRESULT :
STRUCT
	STATUSCODE : OpcUa_StatusCode;
	CONTINUATIONPOINT : OpcUa_ByteString;
	HISTORYDATA : OpcUa_ExtensionObject;
END_STRUCT
END_TYPE

(* ---- OPCUA_HISTORYREADVALUEID.dut ---- *)
TYPE OPCUA_HISTORYREADVALUEID :
STRUCT
	NODEID : OpcUa_NodeId;
	INDEXRANGE : OpcUa_String;
	DATAENCODING : OpcUa_QualifiedName;
	CONTINUATIONPOINT : OpcUa_ByteString;
END_STRUCT
END_TYPE

(* ---- OPCUA_HISTORYUPDATEDETAILS.dut ---- *)
TYPE OPCUA_HISTORYUPDATEDETAILS :
STRUCT
	NODEID : OpcUa_NodeId;
END_STRUCT
END_TYPE

(* ---- OPCUA_HISTORYUPDATEREQUEST.dut ---- *)
TYPE OPCUA_HISTORYUPDATEREQUEST :
STRUCT
	REQUESTHEADER : OpcUa_RequestHeader;
	NOOFHISTORYUPDATEDETAILS : OpcUa_Int32;
	HISTORYUPDATEDETAILS : POINTER TO OpcUa_ExtensionObject;
END_STRUCT
END_TYPE

(* ---- OPCUA_HISTORYUPDATERESPONSE.dut ---- *)
TYPE OPCUA_HISTORYUPDATERESPONSE :
STRUCT
	RESPONSEHEADER : OpcUa_ResponseHeader;
	NOOFRESULTS : OpcUa_Int32;
	RESULTS : POINTER TO OpcUa_HistoryUpdateResult;
	NOOFDIAGNOSTICINFOS : OpcUa_Int32;
	DIAGNOSTICINFOS : POINTER TO OpcUa_DiagnosticInfo;
END_STRUCT
END_TYPE

(* ---- OPCUA_HISTORYUPDATERESULT.dut ---- *)
TYPE OPCUA_HISTORYUPDATERESULT :
STRUCT
	STATUSCODE : OpcUa_StatusCode;
	NOOFOPERATIONRESULTS : OpcUa_Int32;
	OPERATIONRESULTS : POINTER TO OpcUa_StatusCode;
	NOOFDIAGNOSTICINFOS : OpcUa_Int32;
	DIAGNOSTICINFOS : POINTER TO OpcUa_DiagnosticInfo;
END_STRUCT
END_TYPE

(* ---- OPCUA_HISTORYUPDATETYPE.dut ---- *)
TYPE OPCUA_HISTORYUPDATETYPE :
(
	OPCUA_HISTORYUPDATETYPE_INSERT := 1,
	OPCUA_HISTORYUPDATETYPE_REPLACE := 2,
	OPCUA_HISTORYUPDATETYPE_UPDATE := 3,
	OPCUA_HISTORYUPDATETYPE_DELETE := 4
);
END_TYPE

(* ---- OPCUA_IDENTIFIERTYPE.dut ---- *)
TYPE OPCUA_IDENTIFIERTYPE :
(
	OPCUA_IDENTIFIERTYPE_NUMERIC := 0,
	OPCUA_IDENTIFIERTYPE_STRING := 1,
	OPCUA_IDENTIFIERTYPE_GUID := 2,
	OPCUA_IDENTIFIERTYPE_OPAQUE := 3
);
END_TYPE

(* ---- OPCUA_INT.dut ---- *)
TYPE OPCUA_INT : DINT;
END_TYPE

(* ---- OPCUA_INT16.dut ---- *)
TYPE OPCUA_INT16 : INT;
END_TYPE

(* ---- OPCUA_INT32.dut ---- *)
TYPE OPCUA_INT32 : DINT;
END_TYPE

(* ---- OPCUA_INT64.dut ---- *)
TYPE OPCUA_INT64 : LINT;
END_TYPE

(* ---- OPCUA_ISSUEDIDENTITYTOKEN.dut ---- *)
TYPE OPCUA_ISSUEDIDENTITYTOKEN :
STRUCT
	POLICYID : OpcUa_String;
	TOKENDATA : OpcUa_ByteString;
	ENCRYPTIONALGORITHM : OpcUa_String;
END_STRUCT
END_TYPE

(* ---- OPCUA_KEY.dut ---- *)
TYPE OPCUA_KEY :
STRUCT
END_STRUCT
END_TYPE

(* ---- OPCUA_LITERALOPERAND.dut ---- *)
TYPE OPCUA_LITERALOPERAND :
STRUCT
	VALUE : OpcUa_Variant;
END_STRUCT
END_TYPE

(* ---- OPCUA_LOCALIZEDTEXT.dut ---- *)
TYPE OPCUA_LOCALIZEDTEXT :
STRUCT
	LOCALE : OpcUa_String;
	TEXT : OpcUa_String;
END_STRUCT
END_TYPE

(* ---- OPCUA_MDNSDISCOVERYCONFIGURATION.dut ---- *)
TYPE OPCUA_MDNSDISCOVERYCONFIGURATION :
STRUCT
	MDNSSERVERNAME : OpcUa_String;
	NOOFSERVERCAPABILITIES : OpcUa_Int32;
	SERVERCAPABILITIES : POINTER TO OpcUa_String;
END_STRUCT
END_TYPE

(* ---- OPCUA_MESSAGESECURITYMODE.dut ---- *)
TYPE OPCUA_MESSAGESECURITYMODE :
(
	OPCUA_MESSAGESECURITYMODE_INVALID := 0,
	OPCUA_MESSAGESECURITYMODE_NONE := 1,
	OPCUA_MESSAGESECURITYMODE_SIGN := 2,
	OPCUA_MESSAGESECURITYMODE_SIGNANDENCRYPT := 3
);
END_TYPE

(* ---- OPCUA_METHODATTRIBUTES.dut ---- *)
TYPE OPCUA_METHODATTRIBUTES :
STRUCT
	SPECIFIEDATTRIBUTES : OpcUa_UInt32;
	DISPLAYNAME : OpcUa_LocalizedText;
	DESCRIPTION : OpcUa_LocalizedText;
	WRITEMASK : OpcUa_UInt32;
	USERWRITEMASK : OpcUa_UInt32;
	EXECUTABLE : OpcUa_Boolean;
	USEREXECUTABLE : OpcUa_Boolean;
END_STRUCT
END_TYPE

(* ---- OPCUA_MODELCHANGESTRUCTUREDATATYPE.dut ---- *)
TYPE OPCUA_MODELCHANGESTRUCTUREDATATYPE :
STRUCT
	AFFECTED : OpcUa_NodeId;
	AFFECTEDTYPE : OpcUa_NodeId;
	VERB : OpcUa_Byte;
END_STRUCT
END_TYPE

(* ---- OPCUA_MODIFICATIONINFO.dut ---- *)
TYPE OPCUA_MODIFICATIONINFO :
STRUCT
	MODIFICATIONTIME : OpcUa_DateTime;
	UPDATETYPE : OpcUa_HistoryUpdateType;
	USERNAME : OpcUa_String;
END_STRUCT
END_TYPE

(* ---- OPCUA_MODIFYMONITOREDITEMSREQUEST.dut ---- *)
TYPE OPCUA_MODIFYMONITOREDITEMSREQUEST :
STRUCT
	REQUESTHEADER : OpcUa_RequestHeader;
	SUBSCRIPTIONID : OpcUa_UInt32;
	TIMESTAMPSTORETURN : OpcUa_TimestampsToReturn;
	NOOFITEMSTOMODIFY : OpcUa_Int32;
	ITEMSTOMODIFY : POINTER TO OpcUa_MonitoredItemModifyRequest;
END_STRUCT
END_TYPE

(* ---- OPCUA_MODIFYMONITOREDITEMSRESPONSE.dut ---- *)
TYPE OPCUA_MODIFYMONITOREDITEMSRESPONSE :
STRUCT
	RESPONSEHEADER : OpcUa_ResponseHeader;
	NOOFRESULTS : OpcUa_Int32;
	RESULTS : POINTER TO OpcUa_MonitoredItemModifyResult;
	NOOFDIAGNOSTICINFOS : OpcUa_Int32;
	DIAGNOSTICINFOS : POINTER TO OpcUa_DiagnosticInfo;
END_STRUCT
END_TYPE

(* ---- OPCUA_MODIFYSUBSCRIPTIONREQUEST.dut ---- *)
TYPE OPCUA_MODIFYSUBSCRIPTIONREQUEST :
STRUCT
	REQUESTHEADER : OpcUa_RequestHeader;
	SUBSCRIPTIONID : OpcUa_UInt32;
	REQUESTEDPUBLISHINGINTERVAL : OpcUa_Double;
	REQUESTEDLIFETIMECOUNT : OpcUa_UInt32;
	REQUESTEDMAXKEEPALIVECOUNT : OpcUa_UInt32;
	MAXNOTIFICATIONSPERPUBLISH : OpcUa_UInt32;
	PRIORITY : OpcUa_Byte;
END_STRUCT
END_TYPE

(* ---- OPCUA_MODIFYSUBSCRIPTIONRESPONSE.dut ---- *)
TYPE OPCUA_MODIFYSUBSCRIPTIONRESPONSE :
STRUCT
	RESPONSEHEADER : OpcUa_ResponseHeader;
	REVISEDPUBLISHINGINTERVAL : OpcUa_Double;
	REVISEDLIFETIMECOUNT : OpcUa_UInt32;
	REVISEDMAXKEEPALIVECOUNT : OpcUa_UInt32;
END_STRUCT
END_TYPE

(* ---- OPCUA_MONITOREDITEMCREATEREQUEST.dut ---- *)
TYPE OPCUA_MONITOREDITEMCREATEREQUEST :
STRUCT
	ITEMTOMONITOR : OpcUa_ReadValueId;
	MONITORINGMODE : OpcUa_MonitoringMode;
	REQUESTEDPARAMETERS : OpcUa_MonitoringParameters;
END_STRUCT
END_TYPE

(* ---- OPCUA_MONITOREDITEMCREATERESULT.dut ---- *)
TYPE OPCUA_MONITOREDITEMCREATERESULT :
STRUCT
	STATUSCODE : OpcUa_StatusCode;
	MONITOREDITEMID : OpcUa_UInt32;
	REVISEDSAMPLINGINTERVAL : OpcUa_Double;
	REVISEDQUEUESIZE : OpcUa_UInt32;
	FILTERRESULT : OpcUa_ExtensionObject;
END_STRUCT
END_TYPE

(* ---- OPCUA_MONITOREDITEMMODIFYREQUEST.dut ---- *)
TYPE OPCUA_MONITOREDITEMMODIFYREQUEST :
STRUCT
	MONITOREDITEMID : OpcUa_UInt32;
	REQUESTEDPARAMETERS : OpcUa_MonitoringParameters;
END_STRUCT
END_TYPE

(* ---- OPCUA_MONITOREDITEMMODIFYRESULT.dut ---- *)
TYPE OPCUA_MONITOREDITEMMODIFYRESULT :
STRUCT
	STATUSCODE : OpcUa_StatusCode;
	REVISEDSAMPLINGINTERVAL : OpcUa_Double;
	REVISEDQUEUESIZE : OpcUa_UInt32;
	FILTERRESULT : OpcUa_ExtensionObject;
END_STRUCT
END_TYPE

(* ---- OPCUA_MONITOREDITEMNOTIFICATION.dut ---- *)
TYPE OPCUA_MONITOREDITEMNOTIFICATION :
STRUCT
	CLIENTHANDLE : OpcUa_UInt32;
	VALUE : OpcUa_DataValue;
END_STRUCT
END_TYPE

(* ---- OPCUA_MONITORINGMODE.dut ---- *)
TYPE OPCUA_MONITORINGMODE :
(
	OPCUA_MONITORINGMODE_DISABLED := 0,
	OPCUA_MONITORINGMODE_SAMPLING := 1,
	OPCUA_MONITORINGMODE_REPORTING := 2
);
END_TYPE

(* ---- OPCUA_MONITORINGPARAMETERS.dut ---- *)
TYPE OPCUA_MONITORINGPARAMETERS :
STRUCT
	CLIENTHANDLE : OpcUa_UInt32;
	SAMPLINGINTERVAL : OpcUa_Double;
	FILTER : OpcUa_ExtensionObject;
	QUEUESIZE : OpcUa_UInt32;
	DISCARDOLDEST : OpcUa_Boolean;
END_STRUCT
END_TYPE

(* ---- OPCUA_NETWORKGROUPDATATYPE.dut ---- *)
TYPE OPCUA_NETWORKGROUPDATATYPE :
STRUCT
	SERVERURI : OpcUa_String;
	NOOFNETWORKPATHS : OpcUa_Int32;
	NETWORKPATHS : POINTER TO OpcUa_EndpointUrlListDataType;
END_STRUCT
END_TYPE

(* ---- OPCUA_NODEATTRIBUTES.dut ---- *)
TYPE OPCUA_NODEATTRIBUTES :
STRUCT
	SPECIFIEDATTRIBUTES : OpcUa_UInt32;
	DISPLAYNAME : OpcUa_LocalizedText;
	DESCRIPTION : OpcUa_LocalizedText;
	WRITEMASK : OpcUa_UInt32;
	USERWRITEMASK : OpcUa_UInt32;
END_STRUCT
END_TYPE

(* ---- OPCUA_NODECLASS.dut ---- *)
TYPE OPCUA_NODECLASS :
(
	OPCUA_NODECLASS_UNSPECIFIED := 0,
	OPCUA_NODECLASS_OBJECT := 1,
	OPCUA_NODECLASS_VARIABLE := 2,
	OPCUA_NODECLASS_METHOD := 4,
	OPCUA_NODECLASS_OBJECTTYPE := 8,
	OPCUA_NODECLASS_VARIABLETYPE := 16,
	OPCUA_NODECLASS_REFERENCETYPE := 32,
	OPCUA_NODECLASS_DATATYPE := 64,
	OPCUA_NODECLASS_VIEW := 128
);
END_TYPE

(* ---- OPCUA_NODEID.dut ---- *)
TYPE OPCUA_NODEID :
STRUCT
	IDENTIFIERTYPE : OpcUa_IdentifierType;
	NAMESPACEINDEX : OpcUa_UInt16;
	IDENTIFIER : OpcUa_NodeId_anon;
END_STRUCT
END_TYPE

(* ---- OPCUA_NODEID_ANON.dut ---- *)
TYPE OPCUA_NODEID_ANON :
UNION
	NUMERIC : OpcUa_UInt32;
	STRING_CDS : OpcUa_String;
	GUID : POINTER TO OpcUa_Guid;
	BYTESTRING : OpcUa_ByteString;
END_UNION
END_TYPE
